FUNCTION_BLOCK StatusToStringLogPrinterVisitor IMPLEMENTS I_VisitModules, I_VisitSensors
VAR
	stringLog : REFERENCE TO T_MAXSTRING;
END_VAR

METHOD FB_init : BOOL
VAR_INPUT
	bInitRetains : BOOL; // if TRUE, the retain variables are initialized (warm start / cold start)
	bInCopyCode : BOOL;  // if TRUE, the instance afterwards gets moved into the copy code (online change)
	StringLog : REFERENCE TO T_MAXSTRING;
END_VAR
this^.stringLog REF= StringLog;
END_METHOD

METHOD VisitModule
VAR_INPUT
	Module : I_Module;
END_VAR
IF Module.HasError THEN
	RETURN;
END_IF

stringLog := concat(stringLog, '?');
stringLog := concat(stringLog, Module.Name);
stringLog := concat(stringLog, '?');
END_METHOD

METHOD VisitSensor
VAR_INPUT
	Sensor : I_Sensor;
END_VAR
stringLog := concat(stringLog, '<sensor name:=');
stringLog := concat(stringLog, Sensor.Name);
stringLog := concat(stringLog, '>');
END_METHOD

END_FUNCTION_BLOCK

(* stored: Version 1.1.0.1, ProductVersion 3.1.4024.12
   POU StatusToStringLogPrinterVisitor: Id {a759818b-cbed-45ff-a5cc-a58374ec8923}, SpecialFunc None
   Folder Constructor: Id {d1f34462-f595-490f-89ea-583c8e3cae48}
   Method FB_init: Id {3d85aaf6-95c9-4dd6-8ad8-d56f7de56fe1}
   Method VisitModule: Id {6cc7e5cf-f37e-4a04-b972-68d5e1e79e6c}
   Method VisitSensor: Id {413d1d01-5578-4321-ad71-6d4564a94ba0} *)
